//----------------------------------------------------------------------------//
//            Copyright 2018 Rieckermann Engineering Operations               //
//                Automatically Generated File - Do Not Edit                  //
//----------------------------------------------------------------------------//
// Class:       ifbPC1                                                        //
// Description: Instances of PC1                                              //
//                                                                            //
// Vessel ON/OFF pressure control loop with output valve selection.           //
//----------------------------------------------------------------------------//
// Revision history:                                                          //
// Rev By               Date        CC        Note                            //
// 2.1 David Paspa      07-Nov-2018 NA        Simplified by removing valve    //
//                                            selection option performed by   //
//                                            EMC1.                           //
// 2.0 David Paspa      05-Jan-2018 NA        Reboot for S7-1500.             //
// 0.7 Khairul Basar    12-Oct-2009 CC-09/016 IN_REQ_MODE is assigned to      //
//                                            Toggle.                         //
// 0.6 Khairul Basar    16-Sep-2009 CC-09/016 Duplicate Input Parameters      //
//                                            deleted auto/manual both now    //
//                                            using same parameters,Interface //
//                                            FC used for Bumpless changeover.//
// 0.5 Khairul Basar    15-Sep-2009 CC-09/016 PC1 changed.                    //
// 0.4 Khairul Basar    14-Sep-2009 CC-09/016 PC_1110 Setpoint assignment     //
//                                            corrected.                      //
// 0.3 Khairul Basar    09-Sep-2009 CC-09/016 Ref1.                           //
// 0.2 Khairul Basar    01-Sep-2009 CC-09/016 OUT_Qx(BOOL) is changed to      //
//                                            CMD_Qx (INT) & are linked to    //
//                                            POS1valves. Measure variable is //
//                                            lined with PI1 Measure variable.//
//                                            CRIL Interfaced.               //
// 0.1 Khairul Basar    03-Aug-2009           Initial design.                 //
//                                                                            //
// Ref1:Manual and Auto mode is programed.For Manual & auto separate Setpoint,//
// Gas select, & P_CTRL variable created and programmed accordingly.Instance  //
// parameter calls updated."idbPI1".PI_1010.INTERLOCK is linked with NCRIL.  //
//----------------------------------------------------------------------------//
// Index   Instance    Description                                            //
@@TEMPLATE_BEGIN|createInstancesGlobal@@
// @@IDX@@       @@INSTANCE@@      @@DESCRIPTION@@
@@TEMPLATE_END@@
//----------------------------------------------------------------------------//
FUNCTION_BLOCK "ifbPC1"
TITLE = Instances of PC1 pressure controller
{ S7_Optimized_Access := 'TRUE' }
AUTHOR : REO
NAME : ifbPC1
VERSION : 2.1

//----------------------------------------------------------------------------//
// Declare the instance objects of the class:                                 //
//----------------------------------------------------------------------------//
VAR
@@TEMPLATE_BEGIN|createClassNone@@
@@ATTR_BEGIN|numInstances@@
    f : Array[0..@@MAXITEM@@] of "fbPC1";
@@ATTR_END|numInstances@@
@@TEMPLATE_END@@
END_VAR

BEGIN
@@TEMPLATE_BEGIN|createInstances@@
NETWORK
TITLE = Item @@IDX@@ @@INSTANCE@@ : @@DESCRIPTION@@ Critical Interlocks
    //------------------------------------------------------------------------//
    // INSTANCE   INSTANCE   INSTANCE   INSTANCE   INSTANCE   INSTANCE   INST //
    // INSTANCE   INSTANCE   INSTANCE   INSTANCE   INSTANCE   INSTANCE   INST //
    //                                                                        //
    // Get the critical interlock if there is one. If not set alwaysLow:      //
    //------------------------------------------------------------------------//
@@ATTR_BEGIN|CRIL_EXISTS@@
@@ATTR_DEFAULT_BEGIN@@
    A "alwaysLow";
@@ATTR_DEFAULT_END@@
@@ATTR_BEGIN|CRIL_TARGET@@
    A "idbCRIL".p[@@IDXIL@@].INTERLOCK;
@@ATTR_END|CRIL_TARGET@@
@@ATTR_END|CRIL_EXISTS@@
    = #f[@@IDX@@].p.read.mc.CRIL;

NETWORK
TITLE = Item @@IDX@@ @@INSTANCE@@ : @@DESCRIPTION@@ Non-Critical Interlocks
    //------------------------------------------------------------------------//
    // Get the non-critical interlock if there is one. If not set alwaysLow:  //
    //------------------------------------------------------------------------//
@@ATTR_BEGIN|NCRIL_EXISTS@@
@@ATTR_DEFAULT_BEGIN@@
    A "alwaysLow";
@@ATTR_DEFAULT_END@@
@@ATTR_BEGIN|NCRIL_TARGET@@
    A "idbNCRIL".p[@@IDXIL@@].INTERLOCK;
@@ATTR_END|NCRIL_TARGET@@
@@ATTR_END|NCRIL_EXISTS@@
    = #f[@@IDX@@].p.read.mc.NCRIL;

NETWORK
TITLE = Item @@IDX@@ @@INSTANCE@@ : Unique ID
    //------------------------------------------------------------------------//
    // Set the instance unique ID:                                            //
    //------------------------------------------------------------------------//
    L "dbCONST".BLK.ID.@@INSTANCE@@;
    T #f[@@IDX@@].p.read.mc.ME;

NETWORK
TITLE = Item @@IDX@@ @@INSTANCE@@ : Owner ID
    //------------------------------------------------------------------------//
    // Set the instance Owner ID:                                             //
    //------------------------------------------------------------------------//
    L "dbCONST".BLK.ID.@@PARENT@@;
    T #f[@@IDX@@].p.write.mc.OWNER;

@@ATTR_BEGIN|FLOWPATH@@
NETWORK
TITLE = Item @@IDX@@ @@INSTANCE@@ : @@CLASS@@ is a Flowpath device
    //------------------------------------------------------------------------//
    // This class of device is a not a FLOWPATH device where the state must   //
    // equal the command once set by the parent:                              //
    //------------------------------------------------------------------------//
    A "alwaysLow";
    = #f[@@IDX@@].p.read.mc.FLOWPATH;
@@ATTR_END|FLOWPATH@@

NETWORK
TITLE = Item @@IDX@@ @@INSTANCE@@ : Block Read
    //------------------------------------------------------------------------//
    // This block can only reside within this CPU:                            //
    //------------------------------------------------------------------------//
    A "alwaysHigh";
    = #f[@@IDX@@].p.master.read;

NETWORK
TITLE = Item @@IDX@@ @@INSTANCE@@ : Block Write
    //------------------------------------------------------------------------//
    // This block can only be owned by a parent block in this CPU:            //
    //------------------------------------------------------------------------//
    A "alwaysHigh";
    = #f[@@IDX@@].p.master.write;

NETWORK
TITLE = Item @@IDX@@ @@INSTANCE@@ : Set the selected vessel
    //------------------------------------------------------------------------//
    // Set the vessel index number 0,1,2,3 for M1,M2,S1,S2:                   //
    //------------------------------------------------------------------------//
    L @@IDX@@;
    T #f[@@IDX@@].p.write.VESSEL;

NETWORK
TITLE = Item @@IDX@@ @@INSTANCE@@ : Pressure measured value
    //------------------------------------------------------------------------//
    // Set the instance pressure measured value from the PI1:                 //
    //------------------------------------------------------------------------//
@@ATTR_BEGIN|LINK@@
    L @@PILINKIDX@@;         // @@PILINKCLASS@@
    T #f[@@IDX@@].p.link.PRESSURE;
@@ATTR_END|LINK@@

NETWORK
TITLE = Item @@IDX@@ @@INSTANCE@@ : HPCA valve mode and command
    //------------------------------------------------------------------------//
    // Copy the HPCA valve mode and command structures to the PC1 instance:   //
    //------------------------------------------------------------------------//
@@ATTR_BEGIN|LINK@@
    L @@HPCALINKIDX@@;     // @@HPCALINKCLASS@@
    T #f[@@IDX@@].p.link.HPCA;
@@ATTR_END|LINK@@

NETWORK
TITLE = Item @@IDX@@ @@INSTANCE@@ : LPCA valve mode and command
    //------------------------------------------------------------------------//
    // Copy the LPCA valve mode and command structures to the PC1 instance:   //
    //------------------------------------------------------------------------//
@@ATTR_BEGIN|LINK@@
    L @@LPCALINKIDX@@;     // @@LPCALINKCLASS@@
    T #f[@@IDX@@].p.link.LPCA;
@@ATTR_END|LINK@@

NETWORK
TITLE = Item @@IDX@@ @@INSTANCE@@ : VENT valve mode and command
    //------------------------------------------------------------------------//
    // Copy the VENT valve mode and command structures to the PC1 instance:   //
    //------------------------------------------------------------------------//
@@ATTR_BEGIN|LINK@@
    L @@VENTLINKIDX@@;     // @@VENTLINKCLASS@@
    T #f[@@IDX@@].p.link.VENT;
@@ATTR_END|LINK@@

NETWORK
TITLE = Item @@IDX@@ @@INSTANCE@@ : @@DESCRIPTION@@
    //------------------------------------------------------------------------//
    // Call the class function to process each instance:                      //
    //------------------------------------------------------------------------//
    CALL #f[@@IDX@@];

NETWORK
TITLE = Item @@IDX@@ @@INSTANCE@@ : Send the alarm bits to the global DB
    //------------------------------------------------------------------------//
    // Transfer the class event log message bits to the global DB:            //
    //------------------------------------------------------------------------//
    L #f[@@IDX@@].p.read.mc.ALARM;
    T "dbEVENT".alarmBlock.alarm_@@INSTANCE@@;

@@TEMPLATE_END@@

@@TEMPLATE_BEGIN|createInstancesForeign@@
NETWORK
TITLE = Item @@IDX@@ @@INSTANCE@@ : Block Read
    //------------------------------------------------------------------------//
    // This block can only reside in another CPU:                             //
    //------------------------------------------------------------------------//
    A "alwaysLow";
    = #f[@@IDX@@].p.master.read;

@@ATTR_BEGIN|ISOWNED@@
NETWORK
TITLE = Item @@IDX@@ @@INSTANCE@@ : Block Write
    //------------------------------------------------------------------------//
    // This block can only be owned by a parent block in another CPU:         //
    //------------------------------------------------------------------------//
    A "alwaysLow";
    = #f[@@IDX@@].p.master.write;
@@ATTR_END|ISOWNED@@

@@TEMPLATE_END@@

END_FUNCTION_BLOCK
